TYPE stStationCu1 :
STRUCT
	{attribute addProperty Name "Name"}
	Name : STRING := 'Station 1';
	{attribute addProperty Name "Station status"}
	Cu1Enum : stTestEnum;
	{attribute addProperty Name "Time"}
	TimeOfDay: TIME_OF_DAY;
	{attribute addProperty Name "Date"}
    TestDate : DATE;	 
END_STRUCT
END_TYPE

(* stored: Version 1.1.0.1, ProductVersion 3.1.4024.6
   DUT stStationCu1: Id {525f56bc-db0d-0164-0542-83c91861af3d} *)
